PROGRAM MAIN
VAR
	Counter0Inc : DWORD := 1;
	Counter0Read : DWORD; 
	Counter0 : count_mgr_test;
	//Encoder0Read : ULINT;
	Encoder0	:	ST_BisscEncoder;
	EncoderDemand0 : ST_BeamDemand;
	Stepper0	:	ST_Stepper;
	Stepper0EnbP	:	BOOL;
	Stepper0EnbN	:	BOOL;
	
	fbPower	:	MC_Power;
	//fbJog	:	MC_Jog;
	fbHome	:	MC_Home;
	//fbReadStatus	:	MC_ReadStatus;
	fbMoveAbsolute	:	MC_MoveAbsolute;
	fbMoveRelative	:	MC_MoveRelative;
	
END_VAR

//set constants
Encoder0.ncULimit := 170;

//runtime
Counter0(Increment:=Counter0Inc);
Counter0Read := Counter0.CurrentOut;
EncoderDemand0 := FUN_BisscEvaluator(Encoder0);

Stepper0EnbP := Encoder0.encLoc < 1099600;
Stepper0EnbN := Encoder0.encLoc > 460000;

fbPower(Axis:=Stepper0.Axis,Enable:=TRUE,Enable_Positive:=Stepper0EnbP,Enable_Negative:=Stepper0EnbN,Override:=100);

//fbHome(Axis:=Stepper0.Axis,Execute:=TRUE,Position:=4.0,HomingMode:=MC_HomingMode.MC_DefaultHoming);

fbMoveAbsolute(Axis:=Stepper0.Axis,Position:=50.0);

//fbMoveRelative(Axis:=Stepper0.Axis,Execute:=TRUE,Distance:=1);
(*
fbMoveRelative(
	Axis:= , 
	Execute:= , 
	Distance:= , 
	Velocity:= , 
	Acceleration:= , 
	Deceleration:= , 
	Jerk:= , 
	BufferMode:= , 
	Options:= , 
	Done=> , 
	Busy=> , 
	Active=> , 
	CommandAborted=> , 
	Error=> , 
	ErrorID=> );
*)

END_PROGRAM

(* stored: Version 1.1.0.1, ProductVersion 3.1.4020.12
   POU MAIN: Id {c920ae5c-e0ed-41de-acab-e73b0d5cd1a1}, SpecialFunc None *)
